// TIA Portal project "Comunicación entre un PLC y un archivo HTML" (V15.1)

(* hardware
DEVICE "S7-1200 station_1"  S7-1200 Station
   slot 0: "Rack_0"  S7-1200 Rack  Rack  V1.0
   slot 1: "PLC_1"  CPU 1212C AC/DC/Rly  6ES7 212-1BE40-0XB0  V4.2
   slot 2: "AI Energy Meter_1"  SM1238 Energy Meter 480VAC  6ES7 238-5XA32-0XB0  V2.0
   slot 101: "CP 1242-7"  CP 1242-7  6GK7 242-7KX30-0XE0  V1.4
*)

// ===== PLC "PLC_1"  CPU 1212C AC/DC/Rly =====

VAR_GLOBAL   // PLC tag table "Tabla de variables estándar"
   "Motor" AT %Q0.0 : Bool;
   "ValorEscalado" AT %MW66 : Int;
   "Valvula" AT %MW100 : Int;
   "Act_EnergyMeter" AT %I0.1 : Bool;
   "Analog Input" AT %IW64 : Int;
END_VAR

FUNCTION "HTML" : Void   // FC1, LAD
{ S7_Optimized_Access := 'TRUE' }
VERSION : 0.1
   VAR_TEMP
      WebOk : Int;
      Real_V : LReal;
   END_VAR
BEGIN

REGION Network 1
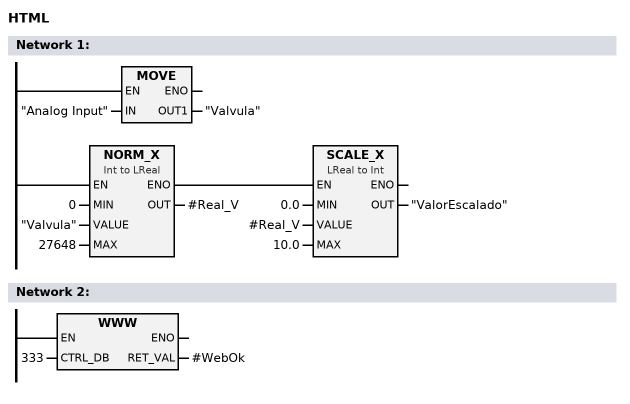
   RUNG wire#powerrail
      Move(in := "Analog Input", out1 => "Valvula")
   END_RUNG
   RUNG wire#powerrail
      { S7_Templates := "[SrcType := Int, DestType := LReal]" } Normalize(min := 0, value := "Valvula", max := 27648, out => #Real_V)
      { S7_Templates := "[SrcType := LReal, DestType := Int]" } Scale(min := 0.0, value := #Real_V, max := 10.0, out => "ValorEscalado")
   END_RUNG
   // the same network as SCL:
   "Valvula" := "Analog Input";
   #Real_V := NORM_X(MIN := 0, VALUE := "Valvula", MAX := 27648);
   "ValorEscalado" := SCALE_X(MIN := 0.0, VALUE := #Real_V, MAX := 10.0);
END_REGION

REGION Network 2
   #WebOk := WWW(CTRL_DB := 333);
END_REGION
END_FUNCTION

ORGANIZATION_BLOCK "Main"   // OB1, LAD, ProgramCycle
TITLE = "Main Program Sweep (Cycle)"
{ S7_Optimized_Access := 'TRUE' }
VERSION : 0.1
   VAR_INPUT
      Initial_Call : Bool;   // Initial call of this OB
      Remanence : Bool;   // =True, if remanent data are available
   END_VAR
BEGIN

REGION Network 1
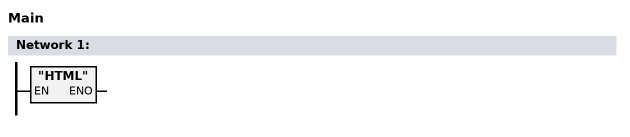
   RUNG wire#powerrail
      "HTML"()
   END_RUNG
   // the same network as SCL:
   "HTML"();
END_REGION
END_ORGANIZATION_BLOCK